// TIA Portal V19 export
DATA_BLOCK "HmiInterface"   // DB110
// stored: Access Published, MemoryReserve 100, Namespace Unit2.Em5
   VAR
      em : "LAF_typeEmInterface";
      jobs : "LAF_typeJobsInterface";
      sequence : "LAF_typeSequenceInterface";
      cm1Vfd208 { S7_SetPoint := 'True'} : "LEXCHANGETRAY_typeRollerVfdInterface";
      cm2Cylinder { S7_SetPoint := 'True'} : "LBC_Simple_typeTwoWayActuatorInterface";
      cm3SignalTM : "LEXCHANGETRAY_typePlasticWorkStationIoSignalInterface";
      cm4Sr1000 { S7_SetPoint := 'True'} : "LEXCHANGETRAY_typeSR1000Interface";
      em5Parameters { S7_SetPoint := 'True'} : "LAF_typePlasticWorkstationEm5ParametersInterface";
   END_VAR
BEGIN
END_DATA_BLOCK
